// TIA Portal V15.1 export
// export: Created 2020-06-12T07:35:52.0380859Z, ExportSetting None, DisplayName Totally Integrated Automation Portal, DisplayVersion V15.1, DisplayName TIA Portal Openness, DisplayVersion V15.1, DisplayName STEP 7 Professional, DisplayVersion V15.1, DisplayName STEP 7 Safety, DisplayVersion V15.1, DisplayName WinCC Advanced, DisplayVersion V15.1
FUNCTION "MELT_Main" : Void   // FC125, FBD
{ S7_Optimized_Access := 'TRUE' }
// stored: SetENOAutomatically False
   VAR_TEMP
      tCondRes : Word;
      tIngot_type : DInt;
      munk_lim_dur : Real;
      tHt_ingot : Bool;
      tConst_lim2_del_off : Bool;
      txxx : Bool;
      tSlagMoltenByPos : Bool;
      tSlagMoltenByEnergy : Bool;
      tReqPrepare : Bool;
      tReqCancel : Bool;
      tReqForceHT : Bool;
      tReqDummy : Bool;
      tReqPause : Bool;
      tReqForseMT : Bool;
      tReqEnd : Bool;
      tReqHT : Bool;
      tReqStop : Bool;
      tVarReal : Real;
      tBool : Bool;
      tSWLock : Bool;
      tMoldIsInserted : Bool;
      tSealingsAreClosed : Bool;
      tReqRestartChk : Bool;
      tMRContEnableByCB : Bool;
      tSWContReqST : Bool;
      tDoStart : Bool;
      tRestartChecks : Bool;
      tHCClamped : Bool;
      tReqReset : Bool;
      tCbIsOn : Bool;
      tReqGasBlow : Bool;
      tCancelReset : Bool;
      tSlagMoltenIsPossible : Bool;
      tReset1 : Bool;
      tSWCLckByDev : Bool;
      tMRContLckByDev : Bool;
      tECRhasFault : Bool;
      tMRLock : Bool;
      tMRContLckByIC : Bool;
      tSWCLckByECR : Bool;
   END_VAR
   VAR_TEMP   // added for the SCL form of the ladder/FBD networks
      _w1 : Bool;
   END_VAR
BEGIN

REGION Network 1: HMI request treat
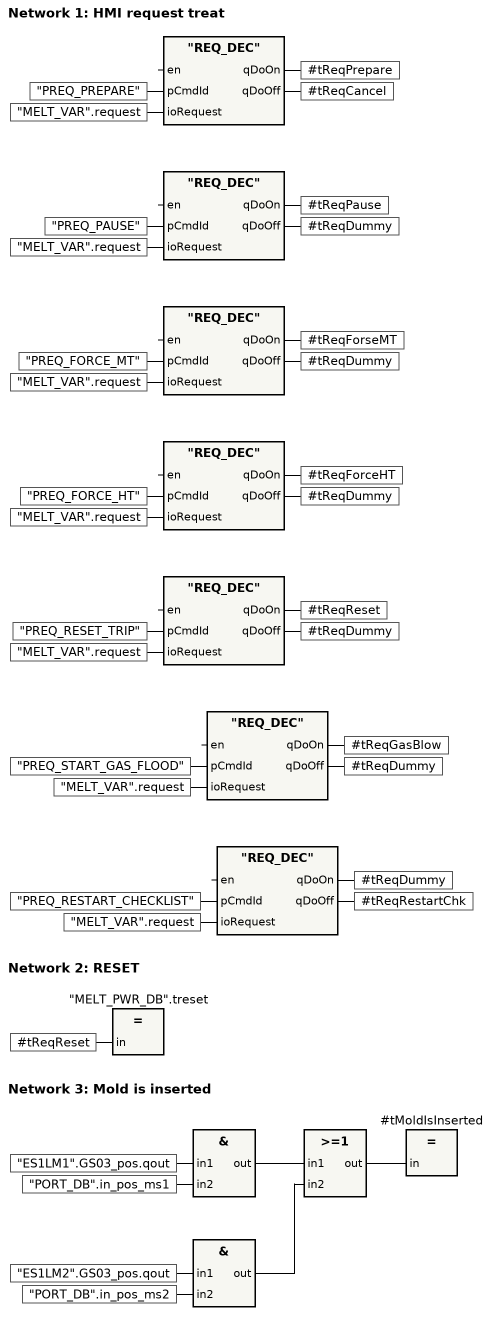
   "REQ_DEC"(pCmdId := "PREQ_PREPARE",
             ioRequest := "MELT_VAR".request,
             qDoOn => #tReqPrepare,
             qDoOff => #tReqCancel);
   "REQ_DEC"(pCmdId := "PREQ_PAUSE", ioRequest := "MELT_VAR".request, qDoOn => #tReqPause, qDoOff => #tReqDummy);
   "REQ_DEC"(pCmdId := "PREQ_FORCE_MT",
             ioRequest := "MELT_VAR".request,
             qDoOn => #tReqForseMT,
             qDoOff => #tReqDummy);
   "REQ_DEC"(pCmdId := "PREQ_FORCE_HT",
             ioRequest := "MELT_VAR".request,
             qDoOn => #tReqForceHT,
             qDoOff => #tReqDummy);
   "REQ_DEC"(pCmdId := "PREQ_RESET_TRIP",
             ioRequest := "MELT_VAR".request,
             qDoOn => #tReqReset,
             qDoOff => #tReqDummy);
   "REQ_DEC"(pCmdId := "PREQ_START_GAS_FLOOD",
             ioRequest := "MELT_VAR".request,
             qDoOn => #tReqGasBlow,
             qDoOff => #tReqDummy);
   "REQ_DEC"(pCmdId := "PREQ_RESTART_CHECKLIST",
             ioRequest := "MELT_VAR".request,
             qDoOn => #tReqDummy,
             qDoOff => #tReqRestartChk);
END_REGION

REGION Network 2: RESET
   "MELT_PWR_DB".treset := #tReqReset;
END_REGION

REGION Network 3: Mold is inserted
   #tMoldIsInserted := ("ES1LM1".GS03_pos.qout AND "PORT_DB".in_pos_ms1) OR ("ES1LM2".GS03_pos.qout AND "PORT_DB".in_pos_ms2);
END_REGION

REGION Network 4: Sealings are ok
   // ! NB PuM: I'm not sure that is really reequired, but...
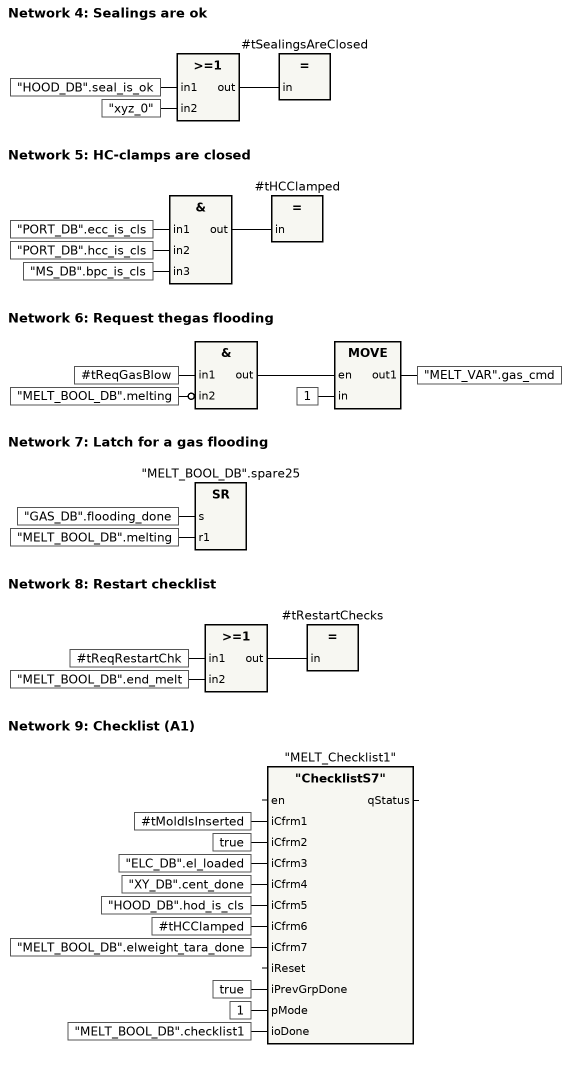
   #tSealingsAreClosed := "HOOD_DB".seal_is_ok OR "xyz_0";
END_REGION

REGION Network 5: HC-clamps are closed
   #tHCClamped := "PORT_DB".ecc_is_cls AND "PORT_DB".hcc_is_cls AND "MS_DB".bpc_is_cls;
END_REGION

REGION Network 6: Request thegas flooding
   IF #tReqGasBlow AND NOT "MELT_BOOL_DB".melting THEN "MELT_VAR".gas_cmd := 1; END_IF;
END_REGION

REGION Network 7: Latch for a gas flooding
   IF "GAS_DB".flooding_done THEN
       "MELT_BOOL_DB".spare25 := TRUE;   // SR flip-flop
   END_IF;
   IF "MELT_BOOL_DB".melting THEN "MELT_BOOL_DB".spare25 := FALSE; END_IF;
END_REGION

REGION Network 8: Restart checklist
   #tRestartChecks := #tReqRestartChk OR "MELT_BOOL_DB".end_melt;
END_REGION

REGION Network 9: Checklist (A1)
   // CHECKLIST:
   // * the mold is inserted
   // * the cooling water pipes are connected
   // * the electrode is loaded/catched
   // * XY platform is in the center
   "MELT_Checklist1"(iCfrm1 := #tMoldIsInserted,   // "ChecklistS7"
                     iCfrm2 := true,
                     iCfrm3 := "ELC_DB".el_loaded,
                     iCfrm4 := "XY_DB".cent_done,
                     iCfrm5 := "HOOD_DB".hod_is_cls,
                     iCfrm6 := #tHCClamped,
                     iCfrm7 := "MELT_BOOL_DB".elweight_tara_done,
                     iPrevGrpDone := true,
                     pMode := 1,
                     ioDone := "MELT_BOOL_DB".checklist1);
END_REGION

REGION Network 10: Checklist (A2)
   // CHECKLIST:
   // * The hood is closed
   // * The HC-clamps are closed
   // * Sealings are activated
   // * The CWS is running (or ready for operation)
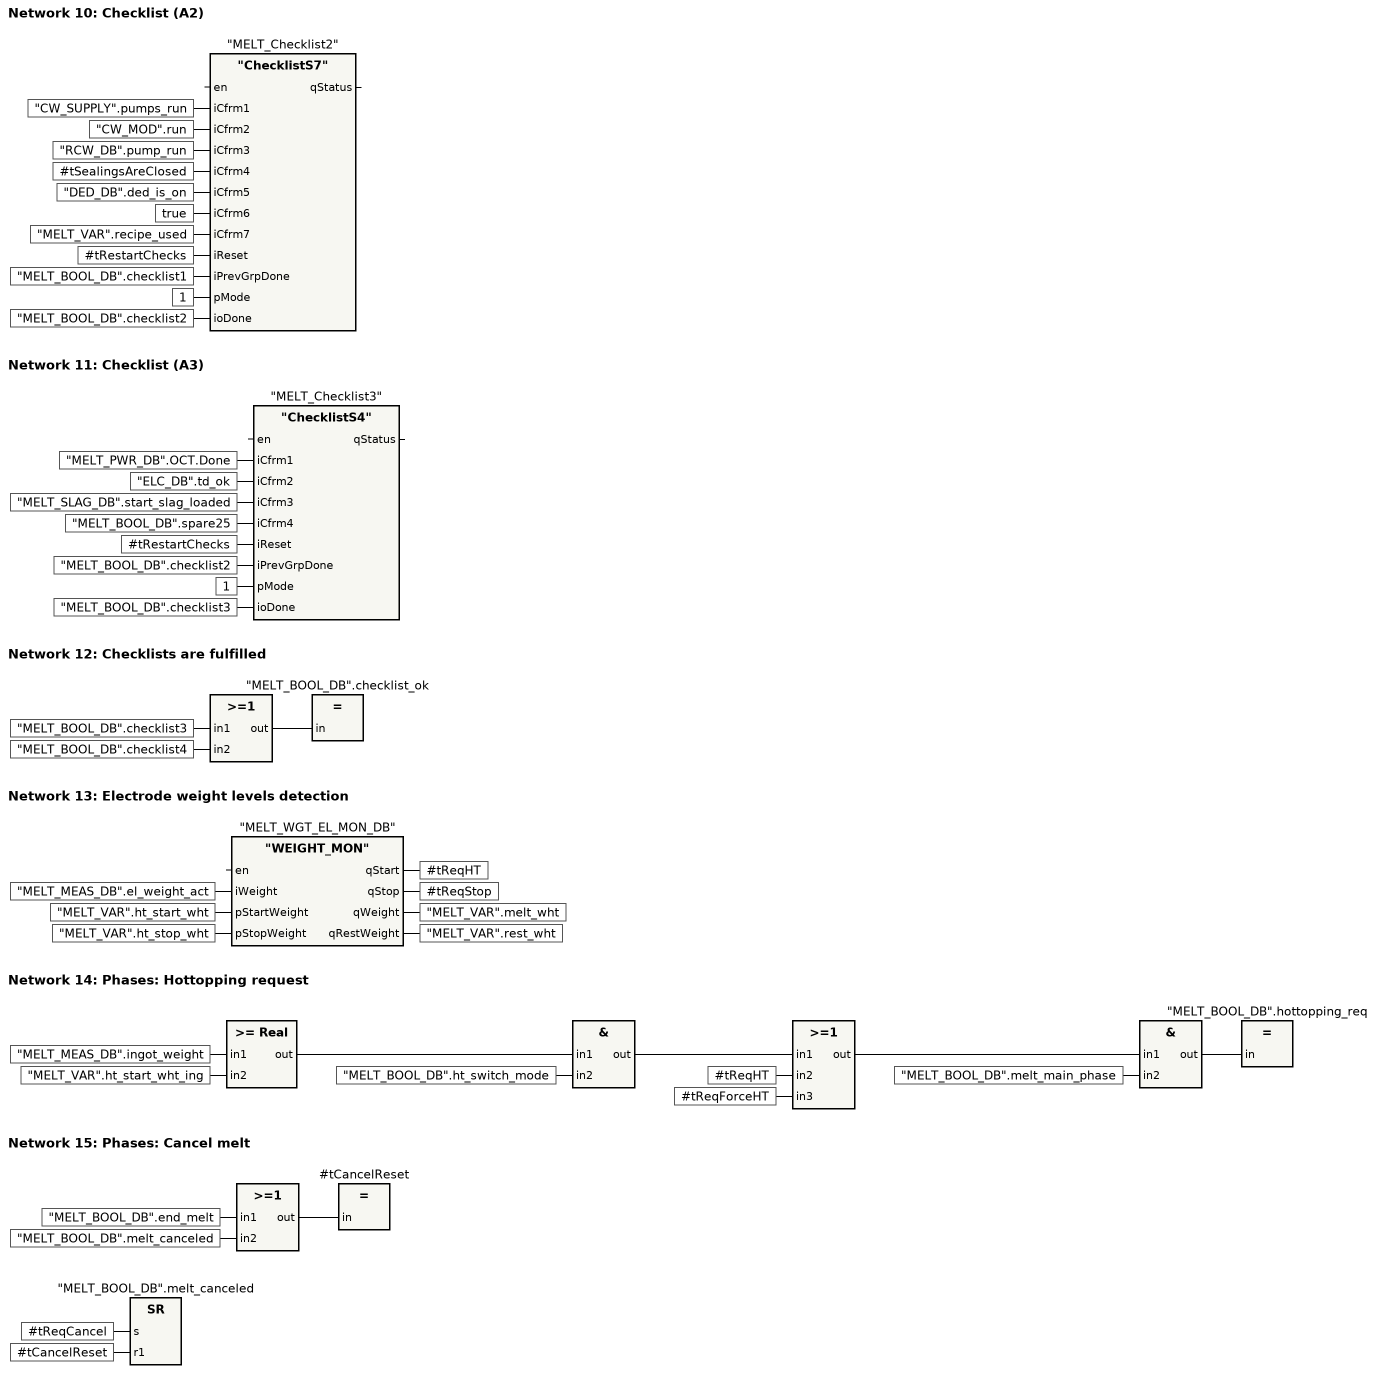
   "MELT_Checklist2"(iCfrm1 := "CW_SUPPLY".pumps_run,   // "ChecklistS7"
                     iCfrm2 := "CW_MOD".run,
                     iCfrm3 := "RCW_DB".pump_run,
                     iCfrm4 := #tSealingsAreClosed,
                     iCfrm5 := "DED_DB".ded_is_on,
                     iCfrm6 := true,
                     iCfrm7 := "MELT_VAR".recipe_used,
                     iReset := #tRestartChecks,
                     iPrevGrpDone := "MELT_BOOL_DB".checklist1,
                     pMode := 1,
                     ioDone := "MELT_BOOL_DB".checklist2);
END_REGION

REGION Network 11: Checklist (A3)
   // CHECKLIST:
   // * The hood is closed
   // * The HC-clamps are closed
   // * Sealings are activated
   // * The CWS is running (or ready for operation)
   "MELT_Checklist3"(iCfrm1 := "MELT_PWR_DB".OCT.Done,   // "ChecklistS4"
                     iCfrm2 := "ELC_DB".td_ok,
                     iCfrm3 := "MELT_SLAG_DB".start_slag_loaded,
                     iCfrm4 := "MELT_BOOL_DB".spare25,
                     iReset := #tRestartChecks,
                     iPrevGrpDone := "MELT_BOOL_DB".checklist2,
                     pMode := 1,
                     ioDone := "MELT_BOOL_DB".checklist3);
END_REGION

REGION Network 12: Checklists are fulfilled
   "MELT_BOOL_DB".checklist_ok := "MELT_BOOL_DB".checklist3 OR "MELT_BOOL_DB".checklist4;
END_REGION

REGION Network 13: Electrode weight levels detection
   "MELT_WGT_EL_MON_DB"(iWeight := "MELT_MEAS_DB".el_weight_act,   // "WEIGHT_MON"
                        pStartWeight := "MELT_VAR".ht_start_wht,
                        pStopWeight := "MELT_VAR".ht_stop_wht,
                        qStart => #tReqHT,
                        qStop => #tReqStop,
                        qWeight => "MELT_VAR".melt_wht,
                        qRestWeight => "MELT_VAR".rest_wht);
END_REGION

REGION Network 14: Phases: Hottopping request
   "MELT_BOOL_DB".hottopping_req := ((("MELT_MEAS_DB".ingot_weight >= "MELT_VAR".ht_start_wht_ing) AND "MELT_BOOL_DB".ht_switch_mode) OR #tReqHT OR #tReqForceHT) AND "MELT_BOOL_DB".melt_main_phase;
END_REGION

REGION Network 15: Phases: Cancel melt
   // TODO:
   #tCancelReset := "MELT_BOOL_DB".end_melt OR "MELT_BOOL_DB".melt_canceled;
   IF #tReqCancel THEN
       "MELT_BOOL_DB".melt_canceled := TRUE;   // SR flip-flop
   END_IF;
   IF #tCancelReset THEN "MELT_BOOL_DB".melt_canceled := FALSE; END_IF;
END_REGION

REGION Network 16: Phases: Stop the melt
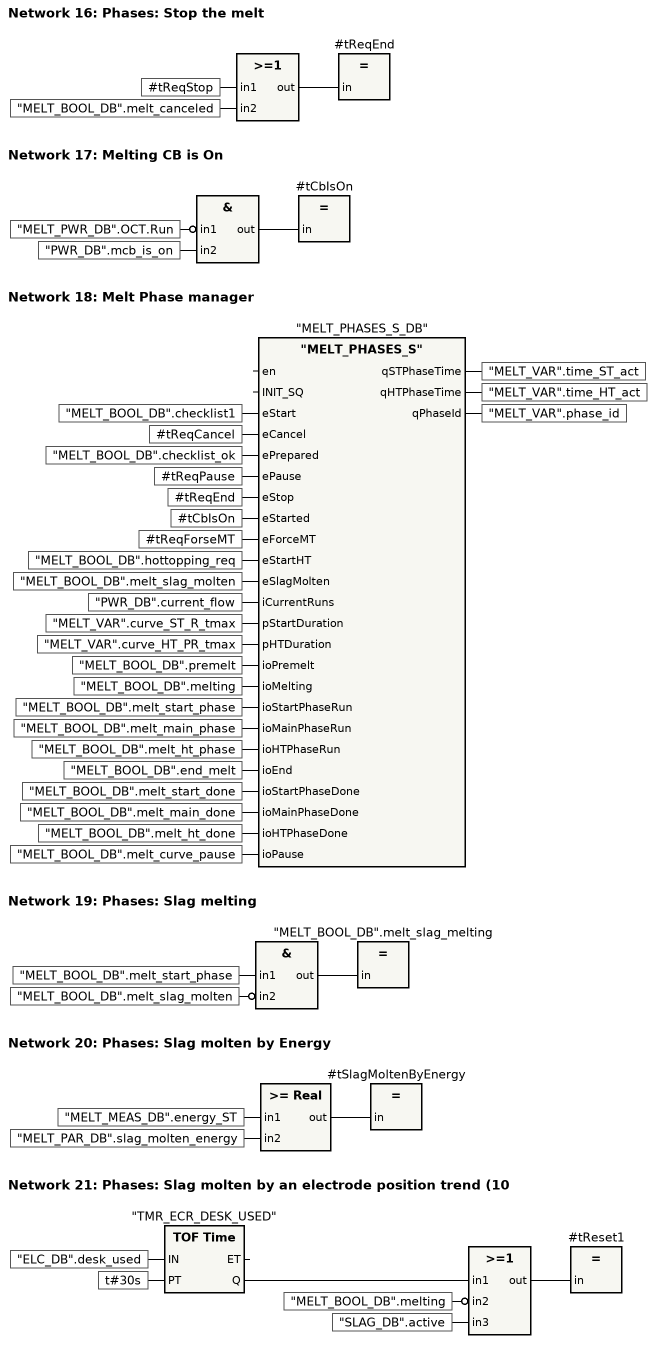
   #tReqEnd := #tReqStop OR "MELT_BOOL_DB".melt_canceled;
END_REGION

REGION Network 17: Melting CB is On
   #tCbIsOn := NOT "MELT_PWR_DB".OCT.Run AND "PWR_DB".mcb_is_on;
END_REGION

REGION Network 18: Melt Phase manager
   "MELT_PHASES_S_DB"(eStart := "MELT_BOOL_DB".checklist1,   // "MELT_PHASES_S"
                      eCancel := #tReqCancel,
                      ePrepared := "MELT_BOOL_DB".checklist_ok,
                      ePause := #tReqPause,
                      eStop := #tReqEnd,
                      eStarted := #tCbIsOn,
                      eForceMT := #tReqForseMT,
                      eStartHT := "MELT_BOOL_DB".hottopping_req,
                      eSlagMolten := "MELT_BOOL_DB".melt_slag_molten,
                      iCurrentRuns := "PWR_DB".current_flow,
                      pStartDuration := "MELT_VAR".curve_ST_R_tmax,
                      pHTDuration := "MELT_VAR".curve_HT_PR_tmax,
                      ioPremelt := "MELT_BOOL_DB".premelt,
                      ioMelting := "MELT_BOOL_DB".melting,
                      ioStartPhaseRun := "MELT_BOOL_DB".melt_start_phase,
                      ioMainPhaseRun := "MELT_BOOL_DB".melt_main_phase,
                      ioHTPhaseRun := "MELT_BOOL_DB".melt_ht_phase,
                      ioEnd := "MELT_BOOL_DB".end_melt,
                      ioStartPhaseDone := "MELT_BOOL_DB".melt_start_done,
                      ioMainPhaseDone := "MELT_BOOL_DB".melt_main_done,
                      ioHTPhaseDone := "MELT_BOOL_DB".melt_ht_done,
                      ioPause := "MELT_BOOL_DB".melt_curve_pause,
                      qSTPhaseTime => "MELT_VAR".time_ST_act,
                      qHTPhaseTime => "MELT_VAR".time_HT_act,
                      qPhaseId => "MELT_VAR".phase_id);
END_REGION

REGION Network 19: Phases: Slag melting
   "MELT_BOOL_DB".melt_slag_melting := "MELT_BOOL_DB".melt_start_phase AND NOT "MELT_BOOL_DB".melt_slag_molten;
END_REGION

REGION Network 20: Phases: Slag molten by Energy
   #tSlagMoltenByEnergy := "MELT_MEAS_DB".energy_ST >= "MELT_PAR_DB".slag_molten_energy;
END_REGION

REGION Network 21: Phases: Slag molten by an electrode position trend (10
   // If operator is using for some reasons the joystick then we need to lock the monitoring for a couple of seconds
   "TMR_ECR_DESK_USED".TOF(IN := "ELC_DB".desk_used, PT := t#30s);
   #tReset1 := "TMR_ECR_DESK_USED".Q OR NOT "MELT_BOOL_DB".melting OR "SLAG_DB".active;
END_REGION

REGION Network 22: Phases: Slag molten by an electrode position trend
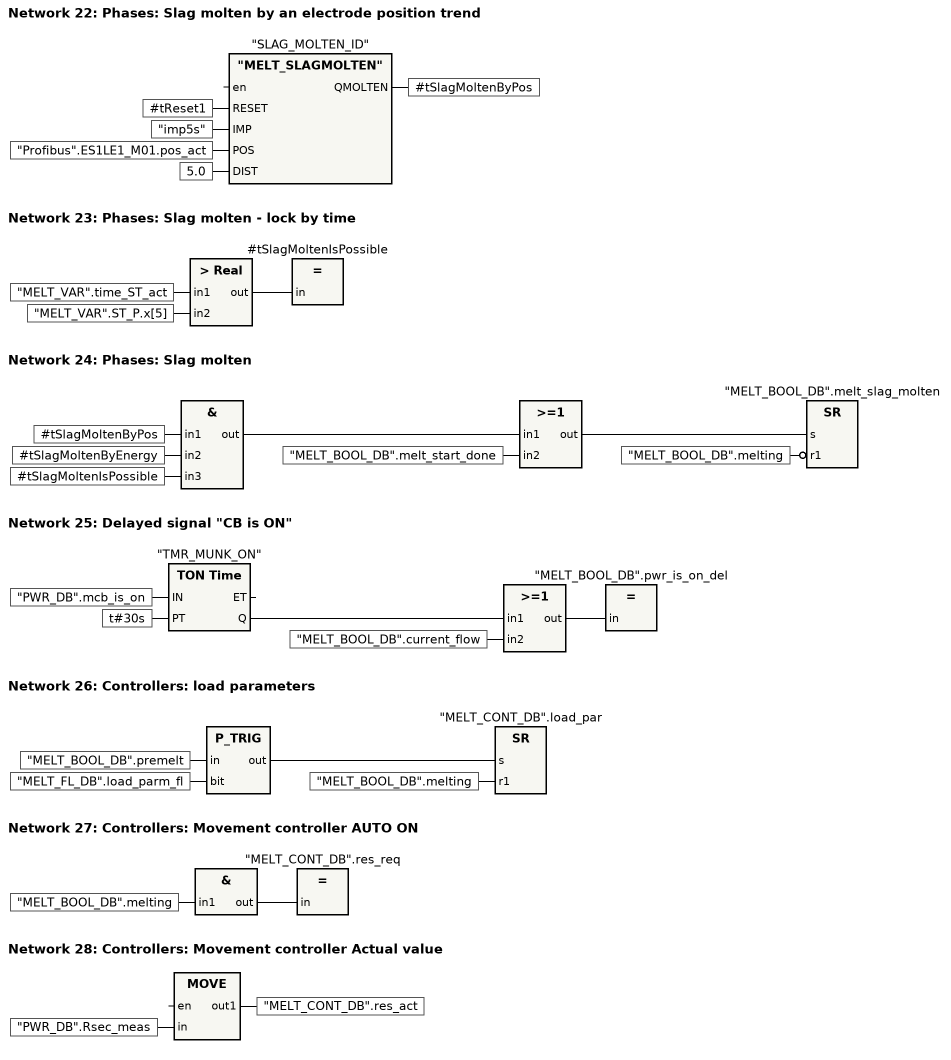
   "SLAG_MOLTEN_ID"(RESET := #tReset1,   // "MELT_SLAGMOLTEN"
                    IMP := "imp5s",
                    POS := "Profibus".ES1LE1_M01.pos_act,
                    DIST := 5.0,
                    QMOLTEN => #tSlagMoltenByPos);
END_REGION

REGION Network 23: Phases: Slag molten - lock by time
   #tSlagMoltenIsPossible := "MELT_VAR".time_ST_act > "MELT_VAR".ST_P.x[5];
END_REGION

REGION Network 24: Phases: Slag molten
   IF (#tSlagMoltenByPos AND #tSlagMoltenByEnergy AND #tSlagMoltenIsPossible) OR "MELT_BOOL_DB".melt_start_done THEN
       "MELT_BOOL_DB".melt_slag_molten := TRUE;   // SR flip-flop
   END_IF;
   IF NOT "MELT_BOOL_DB".melting THEN "MELT_BOOL_DB".melt_slag_molten := FALSE; END_IF;
END_REGION

REGION Network 25: Delayed signal "CB is ON"
   "TMR_MUNK_ON".TON(IN := "PWR_DB".mcb_is_on, PT := t#30s);
   "MELT_BOOL_DB".pwr_is_on_del := "TMR_MUNK_ON".Q OR "MELT_BOOL_DB".current_flow;
END_REGION

REGION Network 26: Controllers: load parameters
   #_w1 := "MELT_BOOL_DB".premelt AND NOT "MELT_FL_DB".load_parm_fl;   // rising edge
   "MELT_FL_DB".load_parm_fl := "MELT_BOOL_DB".premelt;
   IF #_w1 THEN
       "MELT_CONT_DB".load_par := TRUE;   // SR flip-flop
   END_IF;
   IF "MELT_BOOL_DB".melting THEN "MELT_CONT_DB".load_par := FALSE; END_IF;
END_REGION

REGION Network 27: Controllers: Movement controller AUTO ON
   // PuM: Normally this controller is always active, except some situations which can be treat by interlocks
   "MELT_CONT_DB".res_req := "MELT_BOOL_DB".melting;
END_REGION

REGION Network 28: Controllers: Movement controller Actual value
   "MELT_CONT_DB".res_act := "PWR_DB".Rsec_meas;
END_REGION

REGION Network 29: Controllers: Movement controller LOCK
   // PuM/2018-08-02: The controller is always ready, but it could be locked by some circumistanses
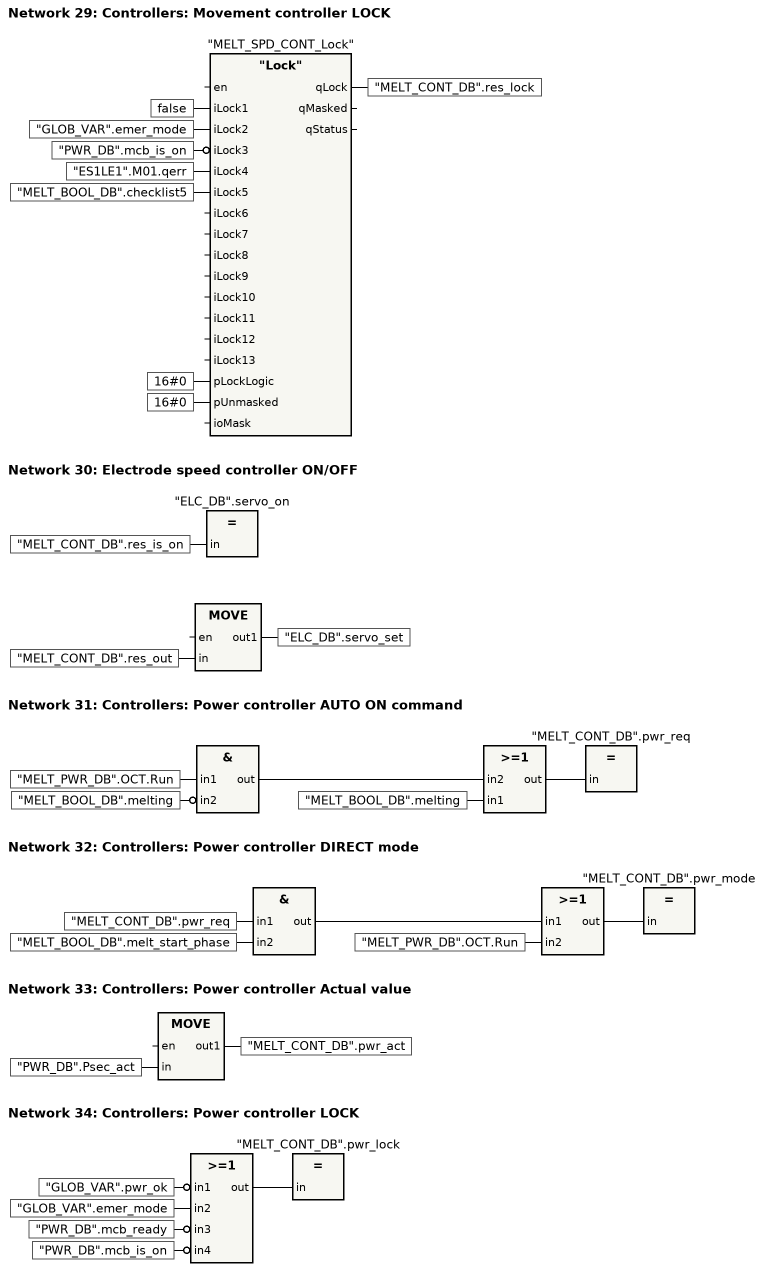
   "MELT_SPD_CONT_Lock"(iLock1 := false,   // "Lock"
                        iLock2 := "GLOB_VAR".emer_mode,
                        iLock3 := NOT "PWR_DB".mcb_is_on,
                        iLock4 := "ES1LE1".M01.qerr,
                        iLock5 := "MELT_BOOL_DB".checklist5,
                        pLockLogic := 16#0,
                        pUnmasked := 16#0,
                        qLock => "MELT_CONT_DB".res_lock);
END_REGION

REGION Network 30: Electrode speed controller ON/OFF
   "ELC_DB".servo_on := "MELT_CONT_DB".res_is_on;
   "ELC_DB".servo_set := "MELT_CONT_DB".res_out;
END_REGION

REGION Network 31: Controllers: Power controller AUTO ON command
   "MELT_CONT_DB".pwr_req := ("MELT_PWR_DB".OCT.Run AND NOT "MELT_BOOL_DB".melting) OR "MELT_BOOL_DB".melting;
END_REGION

REGION Network 32: Controllers: Power controller DIRECT mode
   "MELT_CONT_DB".pwr_mode := ("MELT_CONT_DB".pwr_req AND "MELT_BOOL_DB".melt_start_phase) OR "MELT_PWR_DB".OCT.Run;
END_REGION

REGION Network 33: Controllers: Power controller Actual value
   // "PWR_DB".Psec_act - is filtered value
   "MELT_CONT_DB".pwr_act := "PWR_DB".Psec_act;
END_REGION

REGION Network 34: Controllers: Power controller LOCK
   "MELT_CONT_DB".pwr_lock := NOT "GLOB_VAR".pwr_ok OR "GLOB_VAR".emer_mode OR NOT "PWR_DB".mcb_ready OR NOT "PWR_DB".mcb_is_on;
END_REGION

REGION Network 35: Power controller ON/OFF
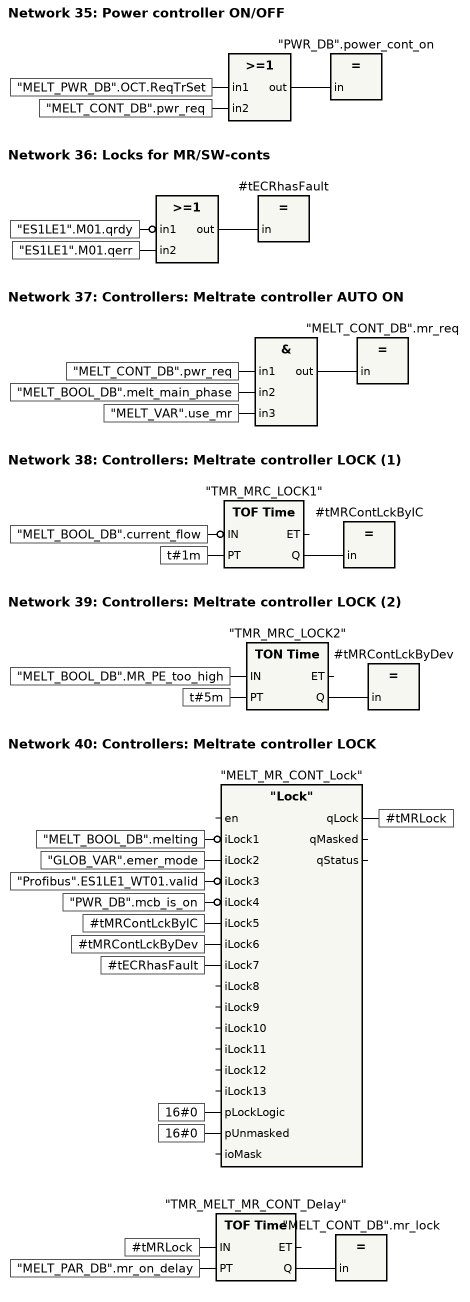
   "PWR_DB".power_cont_on := "MELT_PWR_DB".OCT.ReqTrSet OR "MELT_CONT_DB".pwr_req;
END_REGION

REGION Network 36: Locks for MR/SW-conts
   #tECRhasFault := NOT "ES1LE1".M01.qrdy OR "ES1LE1".M01.qerr;
END_REGION

REGION Network 37: Controllers: Meltrate controller AUTO ON
   "MELT_CONT_DB".mr_req := "MELT_CONT_DB".pwr_req AND "MELT_BOOL_DB".melt_main_phase AND "MELT_VAR".use_mr;
END_REGION

REGION Network 38: Controllers: Meltrate controller LOCK (1)
   "TMR_MRC_LOCK1".TOF(IN := NOT "MELT_BOOL_DB".current_flow, PT := t#1m);
   #tMRContLckByIC := "TMR_MRC_LOCK1".Q;
END_REGION

REGION Network 39: Controllers: Meltrate controller LOCK (2)
   "TMR_MRC_LOCK2".TON(IN := "MELT_BOOL_DB".MR_PE_too_high, PT := t#5m);
   #tMRContLckByDev := "TMR_MRC_LOCK2".Q;
END_REGION

REGION Network 40: Controllers: Meltrate controller LOCK
   "MELT_MR_CONT_Lock"(iLock1 := NOT "MELT_BOOL_DB".melting,   // "Lock"
                       iLock2 := "GLOB_VAR".emer_mode,
                       iLock3 := NOT "Profibus".ES1LE1_WT01.valid,
                       iLock4 := NOT "PWR_DB".mcb_is_on,
                       iLock5 := #tMRContLckByIC,
                       iLock6 := #tMRContLckByDev,
                       iLock7 := #tECRhasFault,
                       pLockLogic := 16#0,
                       pUnmasked := 16#0,
                       qLock => #tMRLock);
   "TMR_MELT_MR_CONT_Delay".TOF(IN := #tMRLock, PT := "MELT_PAR_DB".mr_on_delay);
   "MELT_CONT_DB".mr_lock := "TMR_MELT_MR_CONT_Delay".Q;
END_REGION

REGION Network 41: Controllers: Meltrate controller, Actual value
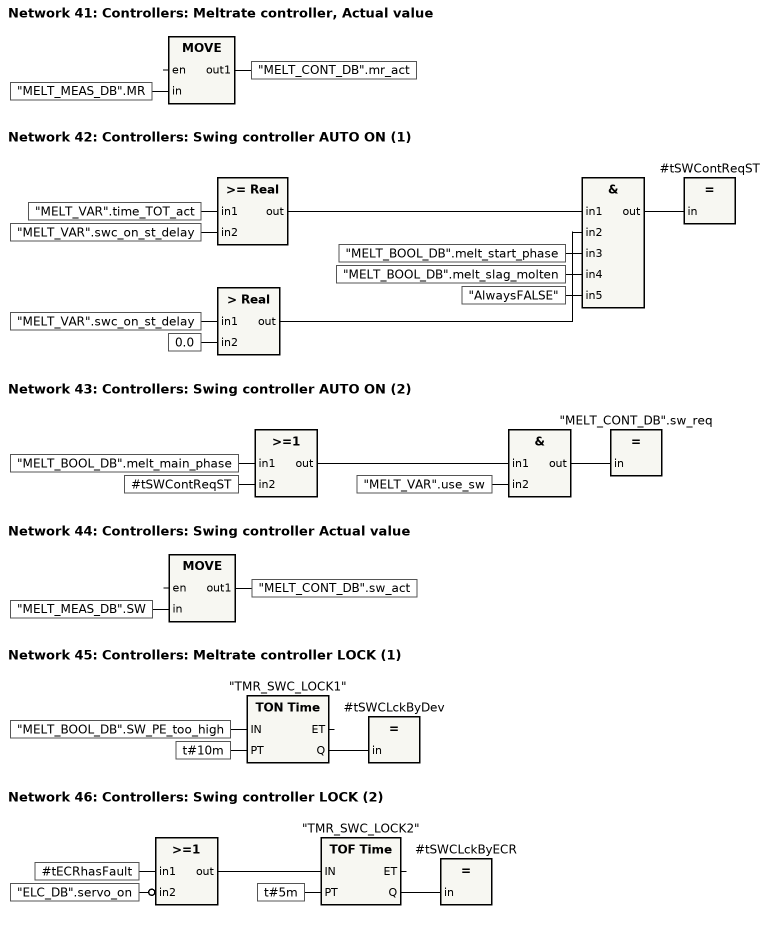
   "MELT_CONT_DB".mr_act := "MELT_MEAS_DB".MR;
END_REGION

REGION Network 42: Controllers: Swing controller AUTO ON (1)
   #tSWContReqST := ("MELT_VAR".time_TOT_act >= "MELT_VAR".swc_on_st_delay) AND ("MELT_VAR".swc_on_st_delay > 0.0) AND "MELT_BOOL_DB".melt_start_phase AND "MELT_BOOL_DB".melt_slag_molten AND "AlwaysFALSE";
END_REGION

REGION Network 43: Controllers: Swing controller AUTO ON (2)
   "MELT_CONT_DB".sw_req := ("MELT_BOOL_DB".melt_main_phase OR #tSWContReqST) AND "MELT_VAR".use_sw;
END_REGION

REGION Network 44: Controllers: Swing controller Actual value
   "MELT_CONT_DB".sw_act := "MELT_MEAS_DB".SW;
END_REGION

REGION Network 45: Controllers: Meltrate controller LOCK (1)
   "TMR_SWC_LOCK1".TON(IN := "MELT_BOOL_DB".SW_PE_too_high, PT := t#10m);
   #tSWCLckByDev := "TMR_SWC_LOCK1".Q;
END_REGION

REGION Network 46: Controllers: Swing controller LOCK (2)
   "TMR_SWC_LOCK2".TOF(IN := #tECRhasFault OR NOT "ELC_DB".servo_on, PT := t#5m);
   #tSWCLckByECR := "TMR_SWC_LOCK2".Q;
END_REGION

REGION Network 47: Controllers: Swing controller LOCK
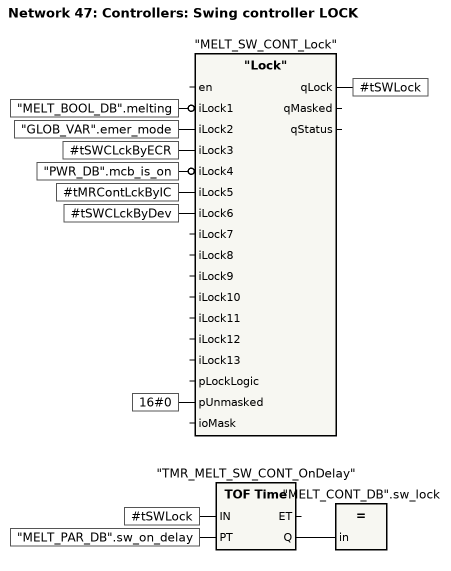
   "MELT_SW_CONT_Lock"(iLock1 := NOT "MELT_BOOL_DB".melting,   // "Lock"
                       iLock2 := "GLOB_VAR".emer_mode,
                       iLock3 := #tSWCLckByECR,
                       iLock4 := NOT "PWR_DB".mcb_is_on,
                       iLock5 := #tMRContLckByIC,
                       iLock6 := #tSWCLckByDev,
                       pUnmasked := 16#0,
                       qLock => #tSWLock);
   "TMR_MELT_SW_CONT_OnDelay".TOF(IN := #tSWLock, PT := "MELT_PAR_DB".sw_on_delay);
   "MELT_CONT_DB".sw_lock := "TMR_MELT_SW_CONT_OnDelay".Q;
END_REGION

REGION Network 48: HMI status
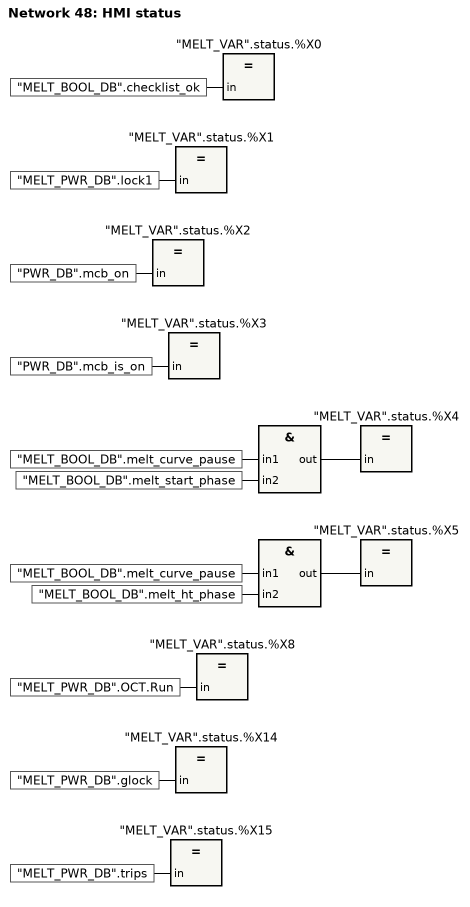
   "MELT_VAR".status.%X0 := "MELT_BOOL_DB".checklist_ok;
   "MELT_VAR".status.%X1 := "MELT_PWR_DB".lock1;
   "MELT_VAR".status.%X2 := "PWR_DB".mcb_on;
   "MELT_VAR".status.%X3 := "PWR_DB".mcb_is_on;
   "MELT_VAR".status.%X4 := "MELT_BOOL_DB".melt_curve_pause AND "MELT_BOOL_DB".melt_start_phase;
   "MELT_VAR".status.%X5 := "MELT_BOOL_DB".melt_curve_pause AND "MELT_BOOL_DB".melt_ht_phase;
   "MELT_VAR".status.%X8 := "MELT_PWR_DB".OCT.Run;
   "MELT_VAR".status.%X14 := "MELT_PWR_DB".glock;
   "MELT_VAR".status.%X15 := "MELT_PWR_DB".trips;
END_REGION
END_FUNCTION
